{attribute 'GeneratedUsingTerminal: ELM2642-0000-0016'}
{attribute addProperty BoxType "ELM2642-0000-0016"}
{attribute addProperty Id "Y1BOOL1Y2BOOL1Y3BOOL1Y4BOOL1"}
{attribute addProperty CRC "2023312392"}
{attribute addProperty Size "4"}
TYPE Outputs_Channel_78994C08 :
STRUCT
	{attribute addProperty Name "Y1"}
	Y1 : BOOL;
	{attribute addProperty Name "Y2"}
	Y2 : BOOL;
	{attribute addProperty Name "Y3"}
	Y3 : BOOL;
	{attribute addProperty Name "Y4"}
	Y4 : BOOL;
END_STRUCT
END_TYPE

(* stored: Version 1.2.0.0, ProductVersion 3.1.4024.9
   DUT Outputs_Channel_78994C08: Id {b5fb0ac1-a32c-49e5-bf37-ad8a557b41b2} *)
